{attribute addProperty BoxType "AT2050-0501-0022"}
{attribute addProperty Id "A_0082_AT2002_5250_0019_AT2002_5250AT2002_C5E5984862678.25"}
{attribute addProperty CRC "2266951156"}
{attribute addProperty SizeInBites "626"}
{attribute addProperty SizeInBytes "78.25"}
TYPE A_0070_AT2050_0501_0022_AT2050_0501_871EEDF4 EXTENDS AT2050_BA5A9548 :
STRUCT
	{attribute addProperty Name "A_0082_AT2002_5250_0019_AT2002_5250"}
	A_0082_AT2002_5250_0019_AT2002_5250 : AT2002_C5E59848;
END_STRUCT
END_TYPE

(* stored: Version 1.2.0.0, ProductVersion 3.1.4024.9
   DUT A_0070_AT2050_0501_0022_AT2050_0501_871EEDF4: Id {6192a37f-48cc-4bef-81dc-786f0d9d73a3} *)
